# EPICS autosave request: iocBoot/iocvxWorks/SGMenu.req
file configMenu.req P=$(P),CONFIG=$(CONFIG)
file softGlue_settings.req  P=$(P),H=$(H)
# for testing remote PV handling
#yyy:userArrayCalc1.DESC
